TYPE TPearlingHead :
	(
		PH_Left := 0,
		PH_Right
	);
END_TYPE

(* stored: Version 1.1.0.1, ProductVersion 3.1.4022.12
   DUT TPearlingHead: Id {99e8532f-6276-4098-bd79-eb3f7e2e1655} *)
